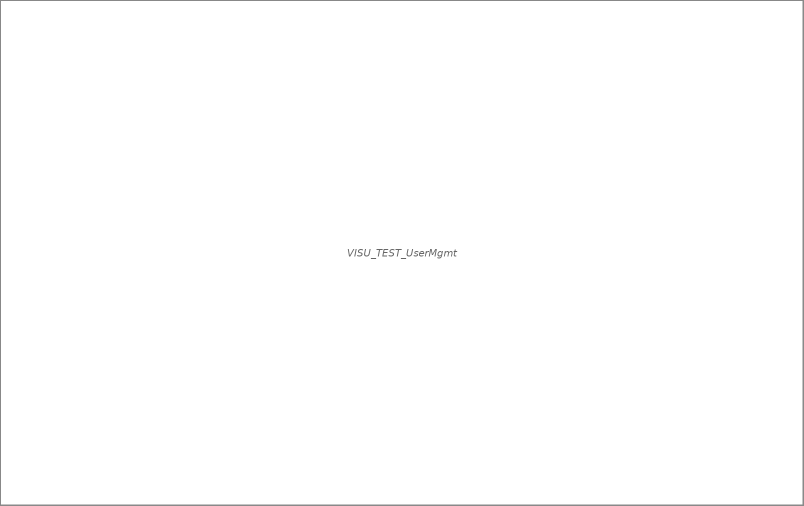
VISUALIZATION VISU_TEST  // 804x506
    TabControl (0,0 804x506)
        shows VISU_TEST_UserMgmt()
        shows ManualControl(stHMI := PRG_TEST_FB_MANUALCONTROLLER.fbManualController.stHMI, fbManualController := PRG_TEST_FB_MANUALCONTROLLER.fbManualController)
        shows ParameterControl()
        [0]: TabTitle=User mgmt
        [1]: TabTitle=ManualControl
        pReferences[1]: fbManualControler=GVL_DevManual.fbManualControler
        [2]: TabTitle=ParameterControl
END_VISUALIZATION

(* stored: Version 1.1.0.1, ProductVersion 3.1.4024.11
   Visu VISU_TEST: Id {57fff5c7-aec8-0420-103f-7f49634e4a49} *)
